{attribute 'pack_mode' := '1'}
TYPE ST_Status :
STRUCT
 RevisionStart, ProtocolVersion, ProfileFingerprint : UDINT;
 State : INT;
 EtherCatOnline, DriveReady, ServoOn, Reserved : BYTE;
 TargetTorqueNm, ActualTorqueNm, SpeedRpm, DcBusV, MotorTempC, BrakeTempC, ServoCurrentA : LREAL;
 ExternalTorqueNm, ExternalSpeedRpm, DutBusV, DutCurrentA : LREAL;
 ValidMask, ErrorCode, InterlockMask, Heartbeat, RevisionEnd : UDINT;
END_STRUCT
END_TYPE

(* stored: Version 1.1.0.1, ProductVersion 3.1.4024.0
   DUT ST_Status: Id {00000000-0000-4000-8000-000000000002} *)
